Fanuc KAREL source: kx00030.KL

-- PROVISIONAL review KL for V770-1; original PC SHA256 113021d648d85d40d083804439d518d7ea45fdc904f108f7c2bdab212d1dab6d
-- Incomplete behavior may be omitted. Consult companion uncertainty JSON. Do not deploy.
PROGRAM KX00030
%NOLOCKGROUP
VAR
  I : INTEGER
  J : INTEGER
  B : BOOLEAN
  F : FILE
  S : STRING[80]
-- UNRESOLVED_DECL P type=000102
BEGIN
  -- UNRESOLVED_PC offsets 5-12; opcodes 9D,23
  -- UNRESOLVED_PC offsets 17-21; opcodes 7F
END KX00030
